// TwinCAT 3 PLC project TcUnit
// ProgramVersion: 3.1.4026.19
// libraries:
//   [AlarmsHandler], * (Marden Edwards)
//   Tc2_Standard, * (Beckhoff Automation GmbH)
//   Tc2_System, * (Beckhoff Automation GmbH)
//   Tc2_TcpIp, * (Beckhoff Automation GmbH)
//   Tc2_Utilities, * (Beckhoff Automation GmbH)
//   TcUnit, * (www.tcunit.org)
// project tree:
//   POUs/ PRG_TEST.TcPOU
//   POUs/TcUnit/FB_Alarm_LogTable/ FB_ALARM_LogTableTests.TcPOU, PRG_FB_ALARM_LogTableManual.TcPOU
//   POUs/Utilities/ PRG_TestsAside.TcPOU
//   / TcUnit_Task.TcTTO
// (motion and I/O tree: see PLC project alarmshandler)
// real-time tasks:
//   TASK TcUnit_Task: cycle T#10ms, priority 10, ADS port 350

CONFIGURATION TcUnit
    RESOURCE PLC ON TwinCAT3
        TASK TcUnit_Task(INTERVAL := T#10ms, PRIORITY := 10);
        PROGRAM PRG_TEST WITH TcUnit_Task : PRG_TEST;
    END_RESOURCE
END_CONFIGURATION

// ---- POUs/PRG_TEST.TcPOU
PROGRAM PRG_TEST
VAR
	fbALARM_Handler		: FB_ALARM_LogTableTests;	
END_VAR

//===================================================
//UNIT TEST EXECUTION

TcUnit.RUN_IN_SEQUENCE();

//===================================================
//MANUAL TEST EXECUTION

PRG_FB_ALARM_LogTableManual();


//PRG_TestsAside();

END_PROGRAM

// ---- POUs/TcUnit/FB_Alarm_LogTable/FB_ALARM_LogTableTests.TcPOU
FUNCTION_BLOCK FB_ALARM_LogTableTests EXTENDS TcUnit.FB_TestSuite

VAR
	
	fbALARM_LogTable		: FB_ALARM_LogTable;	
	
	bResetActive			: BOOL;
	//IN_OUT variables

	stAlarmTable			:	ST_AlarmsTable;
	aAlarms 				: 	ARRAY [0..cMAX_ALARM_GROUP] OF ST_Alarms;
	aAlarmsSettings 		: 	ARRAY [0..cMAX_ALARM_GROUP] OF ST_AlarmSettings;
	stCTDateTime			: 	ST_SYSTEM_DateTime;

END_VAR



//==============================================================
//01.ActiveAlarms
//==============================================================
ActiveAlarms01_aAlarmsActiveSetTrue();
ActiveAlarms02_aAlarmsActiveSetTrue();

//==============================================================
//02.AlarmLogs
//==============================================================
AlarmLogs01_ProperOrder();
AlarmLogs02_ProperOrder();

METHOD INTERNAL ActiveAlarms01_aAlarmsActiveSetTrue
VAR	
	
// 	bResetActive			: BOOL;
// 	//IN_OUT variables
// 
// 	stAlarmTable			:	ST_AlarmsTable;
// 	aAlarms 				: 	ARRAY [0..cMAX_ALARM_GROUP] OF ST_Alarms;
// 	aAlarmsSettings 		: 	ARRAY [0..cMAX_ALARM_GROUP] OF ST_AlarmSettings;
// 	stCTDateTime			: 	ST_SYSTEM_DateTime;
	
END_VAR
// Data init clear
TestInit(aAlarms:= aAlarms, stAlarmTable:= stAlarmTable);
//Change some data for test scenario below
aAlarms[0].nMessage := 16#00000001;

fbALARM_LogTable(
	bResetActive:= bResetActive, 
	stAlarmTable:= stAlarmTable, 
	aAlarms:= aAlarms, 
	aAlarmsSettings:= aAlarmsSettings, 
	stCTDateTime:= stCTDateTime
);

	
IF TcUnit.TEST_ORDERED('ActiveAlarms01_aAlarmsActiveSetTrue') THEN
			
	AssertTrue(	Condition:= (stAlarmTable.aActiveID[0] = TRUE), 
				Message:= 'Active alarm not set'
	);
	AssertTrue(	Condition:= (stAlarmTable.aActiveID[1] = FALSE), 
				Message:= 'No Active alarm set'
	);AssertTrue(	Condition:= (stAlarmTable.aActiveID[33] = FALSE), 
				Message:= 'No Active alarm set'
	);
	AssertTrue(	Condition:= (stAlarmTable.aActiveID[127] = FALSE), 
				Message:= 'No Active alarm set'
	);
	AssertTrue(	Condition:= (stAlarmTable.aActiveID[224] = FALSE), 
				Message:= 'No Active alarm set'
	);

TEST_FINISHED();

END_IF;
END_METHOD

METHOD INTERNAL ActiveAlarms02_aAlarmsActiveSetTrue
VAR	
	
// 	bResetActive			: BOOL;
// 	//IN_OUT variables
// 
// 	stAlarmTable			:	ST_AlarmsTable;
// 	aAlarms 				: 	ARRAY [0..cMAX_ALARM_GROUP] OF ST_Alarms;
// 	aAlarmsSettings 		: 	ARRAY [0..cMAX_ALARM_GROUP] OF ST_AlarmSettings;
// 	stCTDateTime			: 	ST_SYSTEM_DateTime;
	
END_VAR
// Data init clear
TestInit(aAlarms:= aAlarms, stAlarmTable:= stAlarmTable);
//Change some data for test scenario below
aAlarms[1].nMessage := 16#00000001;

fbALARM_LogTable(
	bResetActive:= bResetActive, 
	stAlarmTable:= stAlarmTable, 
	aAlarms:= aAlarms, 
	aAlarmsSettings:= aAlarmsSettings, 
	stCTDateTime:= stCTDateTime
);

	
IF TcUnit.TEST_ORDERED('ActiveAlarms02_aAlarmsActiveSetTrue') THEN
			
	AssertTrue(	Condition:= (stAlarmTable.aActiveID[32] = TRUE), 
				Message:= 'Active alarm not set'
	);
	AssertTrue(	Condition:= (stAlarmTable.aActiveID[0] = FALSE), 
				Message:= 'No Active alarm set'
	);
	AssertTrue(	Condition:= (stAlarmTable.aActiveID[33] = FALSE), 
				Message:= 'No Active alarm set'
	);
	AssertTrue(	Condition:= (stAlarmTable.aActiveID[127] = FALSE), 
				Message:= 'No Active alarm set'
	);
	AssertTrue(	Condition:= (stAlarmTable.aActiveID[224] = FALSE), 
				Message:= 'No Active alarm set'
	);

TEST_FINISHED();

END_IF;
END_METHOD

METHOD INTERNAL AlarmLogs01_ProperOrder
VAR	
	
END_VAR

	
IF TcUnit.TEST_ORDERED('AlarmLogs01_ProperOrder') THEN
	
	// Data init clear
	TestInit(aAlarms:= aAlarms, stAlarmTable:= stAlarmTable);
	//Change some data for test scenario below
	
	aAlarms[0].nMessage := 16#00000001; //alarm no 0
	aAlarms[2].nMessage := 16#00000001; //alarm no 64
	aAlarms[4].nMessage := 16#00000001; //alarm no 128
	
	fbALARM_LogTable(
		bResetActive:= bResetActive, 
		stAlarmTable:= stAlarmTable, 
		aAlarms:= aAlarms, 
		aAlarmsSettings:= aAlarmsSettings, 
		stCTDateTime:= stCTDateTime
	);
			
	AssertEquals_STRING(Actual		:= stAlarmTable.aLogMessages[1],
						Expected	:= 'Alarm No. 128',
						Message		:= 'Alarms not logged properly');

	AssertEquals_STRING(Actual		:= stAlarmTable.aLogMessages[2],
						Expected	:= 'Alarm No. 64',
						Message		:= 'Alarms not logged properly');	

	AssertEquals_STRING(Actual		:= stAlarmTable.aLogMessages[3],
				 		Expected	:= 'Alarm No. 0',
				 		Message		:= 'Alarms not logged properly');	
		 
TEST_FINISHED();

END_IF;
END_METHOD

METHOD INTERNAL AlarmLogs02_ProperOrder
VAR	

END_VAR

	
IF TcUnit.TEST_ORDERED('AlarmLogs02_ProperOrder') THEN
	

	// Data init clear
	TestInit(aAlarms:= aAlarms, stAlarmTable:= stAlarmTable);
	//Change some data for test scenario below
	
	aAlarms[1].nMessage := 16#00000001; //alarm no 32
	aAlarms[3].nMessage := 16#00000001; //alarm no 96
	aAlarms[5].nMessage := 16#00000001; //alarm no 160
	
	fbALARM_LogTable(
		bResetActive	:= bResetActive, 
		stAlarmTable	:= stAlarmTable, 
		aAlarms			:= aAlarms, 
		aAlarmsSettings	:= aAlarmsSettings, 
		stCTDateTime	:= stCTDateTime
	);


			
	AssertEquals_STRING(Actual		:= stAlarmTable.aLogMessages[1],
						Expected	:= 'Alarm No. 160',
						Message		:= 'Alarms not logged properly');

	AssertEquals_STRING(Actual		:= stAlarmTable.aLogMessages[2],
						Expected	:= 'Alarm No. 96',
						Message		:= 'Alarms not logged properly');	

	AssertEquals_STRING(Actual		:= stAlarmTable.aLogMessages[3],
				 		Expected	:= 'Alarm No. 32',
				 		Message		:= 'Alarms not logged properly');	
		 
TEST_FINISHED();

END_IF;
END_METHOD

METHOD PRIVATE TestInit
VAR_IN_OUT
	aAlarms			: ARRAY [0..cMAX_ALARM_GROUP] OF ST_Alarms;
	stAlarmTable	: ST_AlarmsTable;
END_VAR

VAR	
	nI				: INT;
END_VAR

MEMSET(ADR(aAlarms), 16#00, SIZEOF(aAlarms));
MEMSET(ADR(stAlarmTable), 16#00, SIZEOF(stAlarmTable));
stCTDateTime.strHMIDateTime := 'Alarm No.';

FOR nI := 0 TO 255 DO	
	stAlarmTable.aMsgAux[nI].sTextMessage := TO_STRING(nI);		
END_FOR
END_METHOD

END_FUNCTION_BLOCK

// ---- POUs/TcUnit/FB_Alarm_LogTable/PRG_FB_ALARM_LogTableManual.TcPOU
PROGRAM PRG_FB_ALARM_LogTableManual
VAR

	fbALARM_LogTable		: ALARMS.FB_ALARM_LogTable;
	
	bResetActive			: BOOL;
	//IN_OUT variables

	stAlarmTable			:	ST_AlarmsTable;
	aAlarms 				: 	ARRAY [0..cMAX_ALARM_GROUP] OF ST_Alarms;
	aAlarmsSettings 		: 	ARRAY [0..cMAX_ALARM_GROUP] OF ST_AlarmSettings;
	stCTDateTime			: 	ST_SYSTEM_DateTime;
	
	nI	: INT;

END_VAR

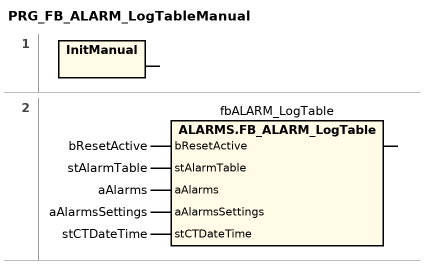
// NETWORK 1
InitManual();

// NETWORK 2
fbALARM_LogTable(
    bResetActive := bResetActive,
    stAlarmTable := stAlarmTable,
    aAlarms := aAlarms,
    aAlarmsSettings := aAlarmsSettings,
    stCTDateTime := stCTDateTime); // ALARMS.FB_ALARM_LogTable

ACTION InitManual:



aAlarms[0].nMessage := 16#00000001;

stCTDateTime.strHMIDateTime := 'Alarm No.';
FOR nI := 0 TO 255 DO	
	stAlarmTable.aMsgAux[nI].sTextMessage := TO_STRING(nI);		
END_FOR
END_ACTION

END_PROGRAM

// ---- POUs/Utilities/PRG_TestsAside.TcPOU
PROGRAM PRG_TestsAside
VAR
	
END_VAR

END_PROGRAM
